// TIA Portal V17 export
// export: Created 2025-03-05T08:02:31.394928Z, ExportSetting WithDefaults, DisplayName Totally Integrated Automation Portal, DisplayVersion V17 Update 8, DisplayName TIA Portal Openness, DisplayVersion V17 Update 8, DisplayName TIA Portal Version Control Interface, DisplayVersion V17, DisplayName SINAMICS Startdrive Advanced, DisplayVersion V17 SP2, DisplayName SINAMICS Startdrive G110M, G120, G120C, G120D, G120P, G115D, DisplayVersion V17 SP2, DisplayName SINAMICS Startdrive G130, G150, S120, S150, SINAMICS MV, S210, DisplayVersion V17 SP2, DisplayName STEP 7 Professional, DisplayVersion V17 Update 8, DisplayName SINUMERIK ONE STEP 7 Toolbox, DisplayVersion V17 Update 12, DisplayName SINUMERIK 840D sl STEP 7 Toolbox, DisplayVersion V17 Update 12, DisplayName STEP 7 Safety, DisplayVersion V17 Update 6, DisplayName WinCC Advanced, DisplayVersion V17 Update 8
TYPE "HMI_MACHINE_OVERVIEW"
// stored: IsFailsafeCompliant false
   STRUCT
      E_STOP_ROBOT : Bool;
      E_STOP_LASER : Bool;
      E_STOP_MAIN_PANEL : Bool;
      E_STOP_MAIN_SAFETY_DOOR : Bool;
      E_STOP_CELL : Bool;
      E_STOP_AUTOMATIC_DOOR : Bool;
      SAFETY_DOOR_L : Bool;
      SAFETY_DOOR_r : Bool;
      MAIN_SAFETY_DOOR : Bool;
      ANALOG_MODE_ON : Bool;
      CONTROL_SPARE_12 : Bool;
      CONTROL_SPARE_13 : Bool;
      CONTROL_SPARE_14 : Bool;
      CONTROL_SPARE_15 : Bool;
      CONTROL_SPARE_16 : Bool;
      CONTROL_SPARE_17 : Bool;
      COMMAND_POWER : DInt;
      REAL_POWER : DInt;
      PYROMETER_ACTUAL_TEMP : Real;
      LENS_HOLDER_FLOW : Real;
      LENS_HOLDER_TEMP : Real;
      ADITIVE_NOZZLE_FLOW : Real;
      ADITIVE_NOZZLE_TEMP : Real;
      DATA7 : DInt;
      DATA8 : DInt;
      DATA9 : Real;
      DATA10 : Real;
      DATA11 : Real;
      DATA12 : Real;
   END_STRUCT;
END_TYPE
